// TIA Portal V15.1 export
// export: Created 2020-12-09T10:45:38.0041669Z, ExportSetting WithDefaults, WithReadOnly, DisplayName Totally Integrated Automation Portal, DisplayVersion V15.1 Update 4, DisplayName TIA Portal Openness, DisplayVersion V15.1, DisplayName SINAMICS Startdrive Advanced, DisplayVersion V15.1 Update3, DisplayName SINAMICS Startdrive G110M, G120, G120C, G120D, G120P, DisplayVersion V15.1 Update3, DisplayName SINAMICS Startdrive G130, G150, S120, S150, SINAMICS MV, S210, DisplayVersion V15.1 Update3, DisplayName STEP 7 Professional, DisplayVersion V15.1 Update 4, DisplayName STEP 7 Safety, DisplayVersion V15.1, DisplayName WinCC Professional, DisplayVersion V15.1 Update 4
DATA_BLOCK "PROAUTOMATOR"   // DB8
{ S7_Optimized_Access := 'TRUE' }
VERSION : 0.1
// stored: AutoNumber true, CodeModifiedDate 2020-12-09T10:16:05.9230189Z, CompileDate 2020-12-09T10:45:34.4747767Z, CreationDate 2020-12-09T09:45:23.3559459Z, DBAccessibleFromOPCUA true, InstanceOfName TYP_PROAUTOMATOR, InstanceOfNumber 15, InstanceOfType UDT, InterfaceModifiedDate 2020-12-09T10:03:08.6573939Z, IsConsistent true, IsKnowHowProtected false, IsOnlyStoredInLoadMemory false, IsWriteProtectedInAS false, ModifiedDate 2020-12-09T10:16:05.9230189Z, ParameterModified 2020-12-09T10:03:08.6573939Z, StructureModified 2020-12-09T10:03:08.6573938Z
"TYP_PROAUTOMATOR"
   // VAR
   //    ST : Struct
   //       Status : "TypStato";
   //    END_STRUCT;
   //    ACTUATORS : Struct
   //       EV : Struct
   //          LimitSwitches : Struct
   //             Home : Bool;
   //             Work : Bool;
   //          END_STRUCT;
   //          Conditions : Struct
   //             Home : Bool;
   //             Work : Bool;
   //          END_STRUCT;
   //          Commands : Struct
   //             Home : Bool;
   //             Work : Bool;
   //          END_STRUCT;
   //          Parameters : "TypValveParameter";
   //       END_STRUCT;
   //    END_STRUCT;
   //    HMI : Struct
   //       FB : Struct
   //          EV : "TypValveFbHmi";
   //       END_STRUCT;
   //       CM : Struct
   //          EV : "TypValveCmHmi";
   //       END_STRUCT;
   //    END_STRUCT;
   //    FEEDBACKS : Struct
   //       EV : "TypValvePosition";
   //    END_STRUCT;
   // END_VAR
BEGIN
END_DATA_BLOCK
